PROGRAM MAIN
VAR
	h1				:	FB_StaticHandler1;
	h2				:	FB_StaticHandler2;
	h3				:	FB_StaticHandler3;
	h_n				:	FB_StaticHandler_n;
	request 		:	STRING	:= 'Hello world!';
	xStartProcess	: 	BOOL;
END_VAR

h1.setNext(h2);
h2.setNext(h3);
h3.setNext(h_n);

(*************************************************************
*************SIMULATION***************************************
***
*** Leave request as "hello world!" for full chain processing
*** or use the string phrases below to interupt the chain.
***
***	Handler 1 - request := 'Handler 1 Interupt';
*** Handler 2 - request := 'Handler 2 Interupt';
*** Handler 3 - request := 'Handler 3 Interupt';
**************************************************************
*************************************************************)

IF xStartProcess THEN
	xStartProcess := FALSE;
	h1.handle(request);
END_IF

END_PROGRAM

(* stored: Version 1.1.0.1, ProductVersion 3.1.4022.16
   POU MAIN: Id {c25706eb-aa71-4377-b614-42f86c7968a7}, SpecialFunc None *)
